ABB RobotStudio station: EX_1_EVAL_ALUM.rspag

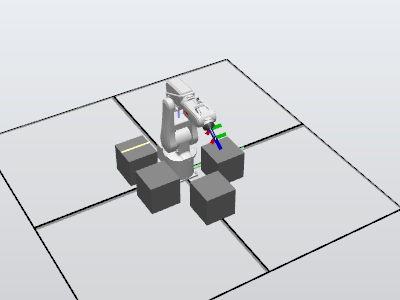
--- station ---
Station EX_1_EVAL (saved by RobotStudio 25.3.11371.0)
Controller IRB120_3_58
  mechanical unit ROB_1: IRB120_3_58__01, 6 joints, base frame (0, 0, 0) mm
Layout (positions relative to the parent item):
  - IRB120_3_58__01 [mechanism, from %ABB.RobotStudio.Models.IRB120%\IRB120_3_58_G_01.rslib] at (0, 0, 0) mm; joint values [0, 0, 0, 0, 0.5236, 0] (rad or m)
  - SC_VentosaV3.3 [protected smart component, left out]
  - Part_1 [part] at (307.45, -105.25, 0) mm, size 200 x 200 x 200 mm
  - Part_2 [part] at (50.03, 129.03, 0) mm, size 200 x 200 x 200 mm
  - Part_3 [part] at (51.63, -340.49, 0) mm, size 200 x 200 x 200 mm
  - Part_4 [part] at (-144.23, -235.54, 200) mm, size 50 x 50 x 50 mm
  - Part_5 [part] at (-244.23, -335.54, 0) mm, size 200 x 200 x 200 mm
  - Piezas [smart component, from Components\piezas.rslib]
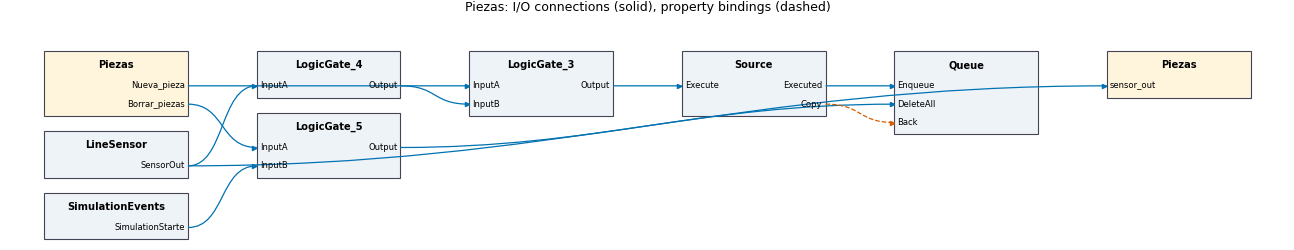
      connections:
        Piezas.Nueva_pieza -> LogicGate_3.InputA
        LineSensor.SensorOut -> LogicGate_4.InputA
        LogicGate_4.Output -> LogicGate_3.InputB
        LogicGate_3.Output -> Source.Execute
        Source.Executed -> Queue.Enqueue
        Piezas.Borrar_piezas -> LogicGate_5.InputA
        SimulationEvents.SimulationStarted -> LogicGate_5.InputB
        LogicGate_5.Output -> Queue.DeleteAll
        LineSensor.SensorOut -> Piezas.sensor_out
        Source.Copy => Queue.Back
    - Source [smart component, from Components\Source.rslib] at (-144.23, -235.54, 200) mm
        properties: Source=Part_4; Copy=(none); Parent=(none); Position=[-0.144228 -0.235544 0.2]; Orientation=[0 0 0]; Transient=false; PhysicsBehavior=-1
    - LineSensor [smart component, from Components\LineSensor.rslib]
        properties: Start=[-0.144228 -0.335544 0.21]; End=[-0.144228 -0.135544 0.21]; Length=0.2; Radius=0; Tag=(none); SensedPart=(none); SensedPoint=[0 0 0]; SenseMultiple=false
      - _sensorPart_ [part], size 0 x 200 x 0 mm
    - LogicGate_3 [smart component, from Components\LogicGate.rslib]
        properties: Operator=AND; Delay=0
    - LogicGate_4 [smart component, from Components\LogicGate.rslib]
        properties: Operator=NOT; Delay=0
    - Queue [smart component, from Components\Queue.rslib]
        properties: Back=(none); Front=(none); Queue=; NumberOfObjects=0
    - SimulationEvents [smart component, from Components\SimulationEvents.rslib]
    - LogicGate_5 [smart component, from Components\LogicGate.rslib]
        properties: Operator=OR; Delay=0
Attachment: SC_VentosaV3.3 is attached to IRB120_3_58__01 / Link6
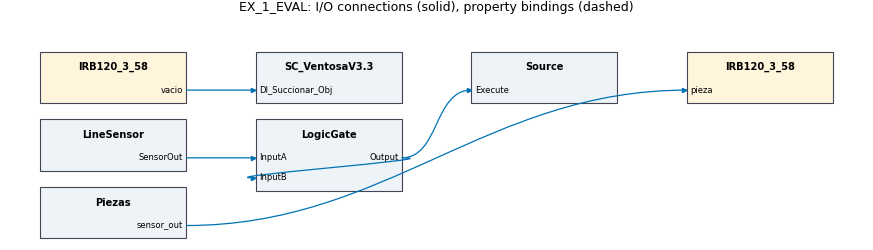
Station logic (signal -> signal, property => property):
  IRB120_3_58.vacio -> SC_VentosaV3.3.DI_Succionar_Objeto
  LineSensor.SensorOut -> LogicGate.InputA
  LogicGate.Output -> LogicGate_2.InputB
  LogicGate_2.Output -> Source.Execute
  Piezas.sensor_out -> IRB120_3_58.pieza

--- Controller Data/IRB120_3_58/RAPID/TASK1/PROGMOD/CalibData.mod ---
MODULE CalibData
    PERS tooldata TCP_Ventosa:=[TRUE,[[0,0,60],[1,0,0,0]],[0.1,[0,0,1],[1,0,0,0],0,0,0]];

ENDMODULE

--- Controller Data/IRB120_3_58/RAPID/TASK1/PROGMOD/Module1.mod ---
MODULE Module1

    VAR num place;

    !***********************************************************
    !
    ! Module:  Module1
    !
    ! Description:
    !   <Insert description here>
    !
    ! Author: windows10
    !
    ! Version: 1.0
    !
    !***********************************************************


    !***********************************************************
    !
    ! Procedure main
    !
    !   This is the entry point of your program
    !
    !***********************************************************
    PROC main()
        !Add your code here

    ENDPROC
ENDMODULE

--- Controller Data/IRB120_3_58/SYSPAR/EIO.cfg ---
EIO:CFG_1.0:6:1::
#
EIO_SIGNAL:

      -Name "vacio" -SignalType "DO" -Access "All"

      -Name "pieza" -SignalType "DI" -Access "All"

      -Name "back" -SignalType "DI" -Access "All"
